FUNCTION_BLOCK EQ_LinearAxis (* Needle lift, a stepper motor through a step and direction driver, with a limit switch at the top (home); equipment IO: owns its IO points, writes the output values its holder sends, reads its inputs every cycle and reports changes *)
  (* Standard: 61499-2 *)
  (* Version 0.1, 2026-09-28, Project contributors, AAU Smart Production Lab *)
  PACKAGE filling;
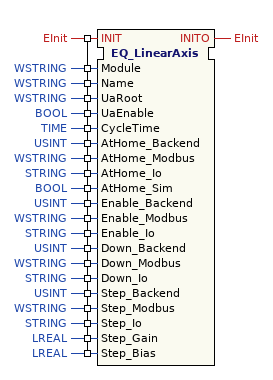
  EVENT_INPUT
    INIT : EInit WITH Module, Name, UaRoot, UaEnable, CycleTime, AtHome_Backend, AtHome_Modbus, AtHome_Io, AtHome_Sim, Enable_Backend, Enable_Modbus, Enable_Io, Down_Backend, Down_Modbus, Down_Io, Step_Backend, Step_Modbus, Step_Io, Step_Gain, Step_Bias;
  END_EVENT
  EVENT_OUTPUT
    INITO : EInit;
  END_EVENT
  VAR_INPUT
    Module : WSTRING;
    Name : WSTRING := "LinearAxis";
    UaRoot : WSTRING;
    UaEnable : BOOL;
    CycleTime : TIME := T#50ms;
    AtHome_Backend : USINT := 2;
    AtHome_Modbus : WSTRING;
    AtHome_Io : STRING;
    AtHome_Sim : BOOL := FALSE;
    Enable_Backend : USINT := 2;
    Enable_Modbus : WSTRING;
    Enable_Io : STRING;
    Down_Backend : USINT := 2;
    Down_Modbus : WSTRING;
    Down_Io : STRING;
    Step_Backend : USINT := 2;
    Step_Modbus : WSTRING;
    Step_Io : STRING;
    Step_Gain : LREAL := 655.35;
    Step_Bias : LREAL := 0.0;
  END_VAR
  (* Group Core: One holder at a time, break before make, all off on release or abort; scanned every CycleTime *)
  (* Group Channels: Local channels to and from the skills (cmd, release, state), the module's state, and the inputs over OPC UA *)
  (* Group Inputs: The equipment's sensors: read every cycle, one block per IO point *)
  (* Group Outputs: The equipment's actuators: written on a change and every cycle, one block per IO point *)
  FBS
    Logic : filling::EL_LinearAxis; {SET_ATTRIBUTE(GroupName, Core)}
    Cycle : iec61499::events::E_CYCLE; {SET_ATTRIBUTE(GroupName, Core)}
    MoveT : iec61499::events::E_DELAY; {SET_ATTRIBUTE(GroupName, Core)}
    Mode : modlib::MOD_StateView; {SET_ATTRIBUTE(GroupName, Channels)}
    SubCmd : iec61499::net::SUBSCRIBE_8(QI := TRUE); {SET_ATTRIBUTE(GroupName, Channels)}
    SubRelease : iec61499::net::SUBSCRIBE_1(QI := TRUE); {SET_ATTRIBUTE(GroupName, Channels)}
    PubState : iec61499::net::PUBLISH_5(QI := TRUE); {SET_ATTRIBUTE(GroupName, Channels)}
    PubUa : iec61499::net::PUBLISH_4; {SET_ATTRIBUTE(GroupName, Channels)}
    In_AtHome : modlib::IO_DI; {SET_ATTRIBUTE(GroupName, Inputs)}
    Out_Enable : modlib::IO_DO; {SET_ATTRIBUTE(GroupName, Outputs)}
    Out_Down : modlib::IO_DO; {SET_ATTRIBUTE(GroupName, Outputs)}
    Out_Step : modlib::IO_AO; {SET_ATTRIBUTE(GroupName, Outputs)}
  END_FBS
  EVENT_CONNECTIONS
    Logic.MOVE_START TO MoveT.START;
    Logic.MOVE_STOP TO MoveT.STOP;
    MoveT.EO TO Logic.MOVE_T;
    INIT TO Logic.INIT;
    Logic.INITO TO Mode.INIT;
    Mode.INITO TO SubCmd.INIT;
    SubCmd.INITO TO SubRelease.INIT;
    SubRelease.INITO TO PubState.INIT;
    PubState.INITO TO PubUa.INIT;
    PubUa.INITO TO In_AtHome.INIT;
    In_AtHome.INITO TO Out_Enable.INIT;
    Out_Enable.INITO TO Out_Down.INIT;
    Out_Down.INITO TO Out_Step.INIT;
    Out_Step.INITO TO Cycle.START;
    Out_Step.INITO TO INITO;
    SubCmd.IND TO Logic.CMD;
    SubRelease.IND TO Logic.RELEASE;
    Mode.CHG TO Logic.MOD_CHG;
    Cycle.EO TO Logic.REFRESH;
    Cycle.EO TO In_AtHome.REQ;
    In_AtHome.CNF TO Logic.SAMPLE;
    Logic.STATE TO PubState.REQ;
    Logic.STATE TO PubUa.REQ;
    Logic.DRIVE TO Out_Enable.REQ;
    Out_Enable.CNF TO Out_Down.REQ;
    Out_Down.CNF TO Out_Step.REQ;
    Out_Step.CNF TO Logic.DRIVEN;
  END_CONNECTIONS
  DATA_CONNECTIONS
    Logic.MoveDT TO MoveT.DT;
    Module TO Logic.Module;
    Name TO Logic.Name;
    UaRoot TO Logic.UaRoot;
    Module TO Mode.Module;
    Logic.IdCmd TO SubCmd.ID;
    Logic.IdRelease TO SubRelease.ID;
    Logic.IdState TO PubState.ID;
    Logic.IdPub TO PubUa.ID;
    UaEnable TO PubUa.QI;
    CycleTime TO Cycle.DT;
    SubCmd.RD_1 TO Logic.C_Holder;
    SubCmd.RD_2 TO Logic.C_Release;
    SubCmd.RD_3 TO Logic.C_Enable;
    SubCmd.RD_4 TO Logic.C_Down;
    SubCmd.RD_5 TO Logic.C_Step;
    SubCmd.RD_6 TO Logic.CE_Step;
    SubCmd.RD_7 TO Logic.C_Move;
    SubCmd.RD_8 TO Logic.C_Goal;
    SubRelease.RD_1 TO Logic.R_Holder;
    Mode.State TO Logic.ModState;
    AtHome_Backend TO In_AtHome.Backend;
    AtHome_Modbus TO In_AtHome.ModbusId;
    AtHome_Io TO In_AtHome.IoName;
    AtHome_Sim TO In_AtHome.SimValue;
    In_AtHome.IN TO Logic.I_AtHome;
    Logic.AtHome TO PubState.SD_1;
    Logic.AtHome TO PubUa.SD_1;
    Logic.ActualPosition TO PubState.SD_2;
    Logic.ActualPosition TO PubUa.SD_2;
    Logic.Homed TO PubState.SD_3;
    Logic.Homed TO PubUa.SD_3;
    Logic.Moving TO PubState.SD_4;
    Logic.Moving TO PubUa.SD_4;
    Logic.Holder TO PubState.SD_5;
    Enable_Backend TO Out_Enable.Backend;
    Enable_Modbus TO Out_Enable.ModbusId;
    Enable_Io TO Out_Enable.IoName;
    Logic.O_Enable TO Out_Enable.OUT;
    Down_Backend TO Out_Down.Backend;
    Down_Modbus TO Out_Down.ModbusId;
    Down_Io TO Out_Down.IoName;
    Logic.O_Down TO Out_Down.OUT;
    Step_Backend TO Out_Step.Backend;
    Step_Modbus TO Out_Step.ModbusId;
    Step_Io TO Out_Step.IoName;
    Logic.O_Step TO Out_Step.OUT;
    Logic.E_Step TO Out_Step.EN;
    Step_Gain TO Out_Step.Gain;
    Step_Bias TO Out_Step.Bias;
  END_CONNECTIONS
END_FUNCTION_BLOCK
